# EPICS autosave request: as/req/modules_F460.req
#FILE... modules_F460.req

file "F460.req", DEVICE=E1:F460
